Staubli VAL3: english.dtx

public string sCancel = "Cancel"
public string sCircular = "Circular"
string sEvtMsg
public string sLinear = "Linear"
public string sListOfMessage[72]
  [0] = "Conveyor calibration utility"
  [1] = "Define conveyor geometry"
  [2] = "Define vision frame"
  [3] = "Define scale factor"
  [4] = "Conveyor overview"
  [5] = "Setup general parameter"
  [6] = "Setup encoder parameter"
  [7] = "Setup detection parameter"
  [8] = "Setup conveyor parameter"
  [9] = "Conveyor Lib."
  [10] = "Encoder Lib."
  [11] = "Detection Lib."
  [12] = "Conveyor type"
  [13] = "Load calibration file"
  [14] = "Conveyor library *\../* is not started, the frame *\../* could not be computed."
  [15] = "Saving successfull"
  [16] = "The library *\../* is going to be deleted, are you sure ?"
  [17] = "Deleting existing conveyor file"
  [18] = "Saving conveyor library"
  [19] = "Saving geometry library"
  [20] = "Do you want to check conveyor geometry?"
  [21] = "Libary name : "
  [22] = "No message pending"
  [23] = "Do you want to define a custom origine for the conveyor's frame"
  [24] = "Error code * while computing the frame associated with the conveyor."
  [25] = "Error while computing vision frame : *"
  [26] = "The digital output selected for the clockSignal parameter is not valid."
  [27] = "The digital output selected for reporting robot motion through the upstream end of conveyor window is not valid"
  [28] = "The digital output selected for reporting robot motion through the downstream end of conveyor window is not valid"
  [30] = "The conveyor library *\../* could not be loaded because of error code * "
  [31] = "The encoder library *\../* could not be loaded because of error code * "
  [32] = "The detection library *\../* could not be loaded because of error code * "
  [33] = "The geometry library *\../* could not be loaded because of error code * "
  [34] = "Your current conveyor library *\../* is beeing saved. Please wait..."
  [35] = "The existing conveyor library *\../* could not be replaced, error code *"
  [36] = "The conveyor library *\../* could not be saved because of error code *"
  [37] = "The geometry library *\../* could not be saved because of error code *"
  [38] = "Wizard>>Couldn't find language file:"
  [40] = "Disable any jog mode"
  [41] = "Disable any jog mode"
  [42] = "Disable the Joint jog mode"
  [43] = "Disable the Frame jog mode"
  [44] = "Disable the Tool jog mode"
  [45] = "Disable the Point jog mode"
  [46] = "Warning, This application requires VAL3 version s7.6.0 or higher"
  [47] = "The valTrack license is not installed or demo period has expired."
  [48] = "Loading your conveyor library *\../* into memory. Please wait..."
  [49] = "Initializing conveyor library"
  [50] = "loading geometry library"
  [51] = "loading encoder library"
  [52] = "loading detection library"
  [53] = "Cannot move to the approach of the current robot position. Please check approach TRSF X=* Y=* Z=*."
  [54] = "Cannot move to the approach of the final destination. Please check approach TRSF X=* Y=* Z=*."
  [55] = "Destination is the out of reach."
  [56] = "Warning: Conveyor not created. Create socket client called 'cognex*', camera's IP address, port 1023, timeout 0. Reload wizard."
  [57] = "Warning: Conveyor not selected. Create socket client called 'cognex*', camera's IP address, port 1023, timeout 0. Reload wizard."
  [58] = "Warning: The output defined as ClkSignal doesn't exist"
  [59] = "Welcome to the Wizard of VALTRACK"
  [60] = "Select/Create a conveyor library"
  [61] = "Warning: Conveyor not created. Create a socket server called 'fromRobot_sk*', port 100*. Reload wizard."
  [62] = "Warning: Conveyor not selected. Create a socket server called 'fromRobot_sk*', port 100*. Reload wizard."
  [63] = "Warning: Message not sent. The socket sent as a parameter is not working. Bad link or device in error."
  [64] = "Warning: Message not sent. Timeout expired. The other robot is not present on the network."
  [65] = "Warning: Message not sent. Timeout expired. The other robot is not working with the detection library 'Socket'."
  [66] = "Warning: Message sent, but the server from the other robot didn't acknowledge reception before expiration of timeout."
  [67] = "VALTRACK"
  [68] = "Warning: Conveyor not created. Edit library Tracking\io\sockets, add to the array of the variable skCognex the index *"
  [69] = "Warning: Conveyor not created. Edit library Tracking\io\sockets, add to the array of the variable skFromRobot the index *"
  [70] = "Warning: Conveyor not selected. Edit library Tracking\io\sockets, add to the array of the variable skCognex the index *"
  [71] = "Warning: Conveyor not selected. Edit library Tracking\io\sockets, add to the array of the variable skFromRobot the index *"
public string sMenu[60]
  [0] = "; ; ; OK ; ; CANCEL"
  [1] = "; ; ; OK"
  [4] = "PREVIOUS UNDO SELECT ; AVERAGE ; NEXT CANCEL"
  [5] = "PREVIOUS ; ; ADJUST ; ; NEXT CANCEL"
  [6] = "PREVIOUS HERE MOVE ; ; ; NEXT CANCEL"
  [7] = "PREVIOUS HERE ; ; ; ; NEXT CANCEL"
  [8] = "PREVIOUS ; ; ; ; ; ; CANCEL"
  [9] = "; ; ; ; ; ; NEXT CANCEL"
  [10] = "; NEW DUPLICATE SELECT ; DELETE  ; QUIT"
  [11] = "; NEW ; ; ; ; ; QUIT"
  [12] = "; ; ; SELECT ; ; ; CANCEL"
  [13] = "PREVIOUS ; ; SELECT ; ; ; CANCEL"
  [14] = "; HERE MOVE ; ; VIEW NEXT CANCEL"
  [15] = "; HERE ; ; ; VIEW NEXT CANCEL"
  [16] = "PREVIOUS HERE MOVE ; ; VIEW NEXT CANCEL"
  [17] = "PREVIOUS HERE ; ; ; VIEW NEXT CANCEL"
  [18] = "PREVIOUS ; ; ; ; ; NEXT CANCEL"
  [19] = "PREVIOUS NEW ; SELECT ; ; ; CANCEL"
  [20] = "PREVIOUS NEW ; ; ; ; ; CANCEL"
  [21] = "; ; YES ; ; ; NO"
  [22] = "; ; YES ; ; ;  NO CANCEL"
  [23] = "; LATCH ; ; ; ; NEXT CANCEL"
  [50] = "F1: Define Scale factor"
  [51] = "F2: Conveyor geometry"
  [52] = "F3: Define Sensor Distance"
  [53] = "F4: Conveyor Diagnostic"
  [54] = "F5: Complete calibration sequence"
  [55] = "F8: Quit"
public string sNONE = "none"
public string sNOTDEFINED = "Not defined"
public string sNo = "No"
public string sOptionTitle
public string sYes = "Yes"
public trsf trTrsf[4]
public mdesc mNomSpeed = {blend=off}
